// TIA Portal project "Project10" (V15.1)

(* hardware
DEVICE "S71500/ET200MP station_1"  S7-1500 station
   slot 0: "Rail_0"  Rack  6ES7 590-1***0-0AA0
   slot 1: "PLC_1"  CPU 1511C-1 PN  6ES7 511-1CK00-0AB0  V2.6
      slot 3: "CPU display_1"  6ES7591-1AA00-0AA0
DEVICE "HMI_1"  TP700 Comfort
   slot 0: "HMI_1"  TP700 Comfort  6AV2 124-0GC01-0AX0  15.1.0.0
   slot 1: "HMI_RT_1"  TP700 Comfort  6AV2 124-0GC01-0AX0  15.1.0.0
   slot 5: "HMI_1.IE_CP_1"  PROFINET Interface  15.0.1.0
      slot 1: "PROFINET Interface_1"  PROFINET Interface
         slot 1: "Port_1"  Port
         slot 2: "Port_2"  Port
   slot 7: "HMI_1.MPI/DP_CP_1"  MPI/DP Interface  15.0.1.0
*)

// ===== PLC "PLC_1"  CPU 1511C-1 PN =====

VAR_GLOBAL   // PLC tag table "Default tag table"
   "Allow_instrybutor" AT %M500.5 : Bool;
   "Tag_1" AT %I0.1 : Bool;
   "tag_test" AT %I0.2 : Bool;
   "Tag_2" AT %M1.1 : Bool;
END_VAR

DATA_BLOCK "CompareLoginPassword_DB"   // DB1
{ S7_Optimized_Access := 'TRUE' }
VERSION : 0.1
// stored: InstanceOfName CompareLoginPassword
"CompareLoginPassword"
BEGIN
END_DATA_BLOCK

DATA_BLOCK "HMI"   // DB2
{ S7_Optimized_Access := 'TRUE' }
VERSION : 0.1
   VAR
      User_Struct_1 : Struct
         login : Int := 1111;
         password : Int := 1111;
         fuel_amount : Int := 50;
      END_STRUCT;
      User_Struct_2 : Struct
         login : Int := 555;
         password : Int := 555;
         fuel_amount : Int;
      END_STRUCT;
      User_Struct_3 : Struct
         login : Int := 352;
         password : Int := 523;
         fuel_amount : Int;
      END_STRUCT;
      User_Struct_4 : Struct
         login : Int := 568;
         password : Int := 8568;
         fuel_amount : Int;
      END_STRUCT;
      User_Struct_5 : Struct
         login : Int := 5665;
         password : Int := 6555;
         fuel_amount : Int;
      END_STRUCT;
      User_Struct_6 : Struct
         login : Int := 5343;
         password : Int := 1234;
         fuel_amount : Int;
      END_STRUCT;
      User_Struct_7 : Struct
         login : Int := 3321;
         password : Int := 5453;
         fuel_amount : Int;
      END_STRUCT;
      User_Struct_8 : Struct
         login : Int := 6233;
         password : Int := 6433;
         fuel_amount : Int;
      END_STRUCT;
      User_Struct_9 : Struct
         login : Int := 612;
         password : Int := 1253;
         fuel_amount : Int;
      END_STRUCT;
      User_Struct_10 : Struct
         login : Int := 1213;
         password : Int := 1235;
         fuel_amount : Int;
      END_STRUCT;
      HMI_Login_Int : Int;
      HMI_Password_Int : Int;
      HMI_Button_Pressed : Bool;
      HMI_Access_Granted : Bool;
      HMI_Fuel_Amount : Int;
      HMI_Screen_Access : Int;
      filled_value : Int;
      WWW_Tag : Int;
      memory : Int := 1500;
   END_VAR
BEGIN
END_DATA_BLOCK

DATA_BLOCK "instrybutor_DB"   // DB4
{ S7_Optimized_Access := 'TRUE' }
VERSION : 0.1
// stored: InstanceOfName instrybutor
"instrybutor"
BEGIN
END_DATA_BLOCK

// folder: System blocks/Program resources

DATA_BLOCK "IEC_Timer_0_DB"   // DB3
{ S7_Optimized_Access := 'TRUE' }
AUTHOR : Simatic
FAMILY : IEC
NAME : IEC_TMR
VERSION : 1.0
// stored: InstanceOfName IEC_TIMER
"IEC_TIMER"
BEGIN
END_DATA_BLOCK

// folder: (top level)

FUNCTION_BLOCK "CompareLoginPassword"   // FB1, LAD
{ S7_Optimized_Access := 'TRUE' }
VERSION : 0.1
BEGIN

REGION Network 1
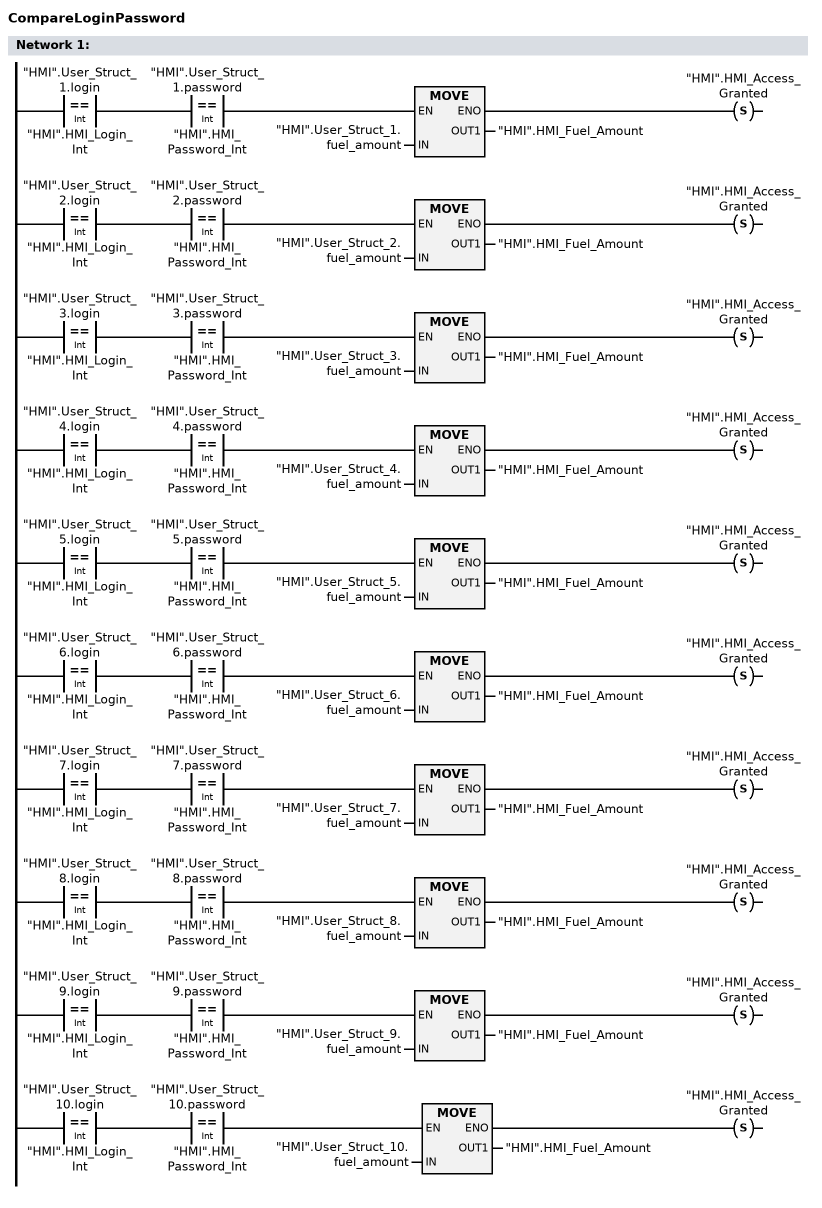
   RUNG wire#powerrail
      { S7_Templates := "SrcType := Int" } EQ_Contact(in1 := "HMI".User_Struct_1.login, in2 := "HMI".HMI_Login_Int)
      { S7_Templates := "SrcType := Int" } EQ_Contact(in1 := "HMI".User_Struct_1.password, in2 := "HMI".HMI_Password_Int)
      Move(in := "HMI".User_Struct_1.fuel_amount, out1 => "HMI".HMI_Fuel_Amount)
      S_Coil( "HMI".HMI_Access_Granted )
   END_RUNG
   RUNG wire#powerrail
      { S7_Templates := "SrcType := Int" } EQ_Contact(in1 := "HMI".User_Struct_2.login, in2 := "HMI".HMI_Login_Int)
      { S7_Templates := "SrcType := Int" } EQ_Contact(in1 := "HMI".User_Struct_2.password, in2 := "HMI".HMI_Password_Int)
      Move(in := "HMI".User_Struct_2.fuel_amount, out1 => "HMI".HMI_Fuel_Amount)
      S_Coil( "HMI".HMI_Access_Granted )
   END_RUNG
   RUNG wire#powerrail
      { S7_Templates := "SrcType := Int" } EQ_Contact(in1 := "HMI".User_Struct_3.login, in2 := "HMI".HMI_Login_Int)
      { S7_Templates := "SrcType := Int" } EQ_Contact(in1 := "HMI".User_Struct_3.password, in2 := "HMI".HMI_Password_Int)
      Move(in := "HMI".User_Struct_3.fuel_amount, out1 => "HMI".HMI_Fuel_Amount)
      S_Coil( "HMI".HMI_Access_Granted )
   END_RUNG
   RUNG wire#powerrail
      { S7_Templates := "SrcType := Int" } EQ_Contact(in1 := "HMI".User_Struct_4.login, in2 := "HMI".HMI_Login_Int)
      { S7_Templates := "SrcType := Int" } EQ_Contact(in1 := "HMI".User_Struct_4.password, in2 := "HMI".HMI_Password_Int)
      Move(in := "HMI".User_Struct_4.fuel_amount, out1 => "HMI".HMI_Fuel_Amount)
      S_Coil( "HMI".HMI_Access_Granted )
   END_RUNG
   RUNG wire#powerrail
      { S7_Templates := "SrcType := Int" } EQ_Contact(in1 := "HMI".User_Struct_5.login, in2 := "HMI".HMI_Login_Int)
      { S7_Templates := "SrcType := Int" } EQ_Contact(in1 := "HMI".User_Struct_5.password, in2 := "HMI".HMI_Password_Int)
      Move(in := "HMI".User_Struct_5.fuel_amount, out1 => "HMI".HMI_Fuel_Amount)
      S_Coil( "HMI".HMI_Access_Granted )
   END_RUNG
   RUNG wire#powerrail
      { S7_Templates := "SrcType := Int" } EQ_Contact(in1 := "HMI".User_Struct_6.login, in2 := "HMI".HMI_Login_Int)
      { S7_Templates := "SrcType := Int" } EQ_Contact(in1 := "HMI".User_Struct_6.password, in2 := "HMI".HMI_Password_Int)
      Move(in := "HMI".User_Struct_6.fuel_amount, out1 => "HMI".HMI_Fuel_Amount)
      S_Coil( "HMI".HMI_Access_Granted )
   END_RUNG
   RUNG wire#powerrail
      { S7_Templates := "SrcType := Int" } EQ_Contact(in1 := "HMI".User_Struct_7.login, in2 := "HMI".HMI_Login_Int)
      { S7_Templates := "SrcType := Int" } EQ_Contact(in1 := "HMI".User_Struct_7.password, in2 := "HMI".HMI_Password_Int)
      Move(in := "HMI".User_Struct_7.fuel_amount, out1 => "HMI".HMI_Fuel_Amount)
      S_Coil( "HMI".HMI_Access_Granted )
   END_RUNG
   RUNG wire#powerrail
      { S7_Templates := "SrcType := Int" } EQ_Contact(in1 := "HMI".User_Struct_8.login, in2 := "HMI".HMI_Login_Int)
      { S7_Templates := "SrcType := Int" } EQ_Contact(in1 := "HMI".User_Struct_8.password, in2 := "HMI".HMI_Password_Int)
      Move(in := "HMI".User_Struct_8.fuel_amount, out1 => "HMI".HMI_Fuel_Amount)
      S_Coil( "HMI".HMI_Access_Granted )
   END_RUNG
   RUNG wire#powerrail
      { S7_Templates := "SrcType := Int" } EQ_Contact(in1 := "HMI".User_Struct_9.login, in2 := "HMI".HMI_Login_Int)
      { S7_Templates := "SrcType := Int" } EQ_Contact(in1 := "HMI".User_Struct_9.password, in2 := "HMI".HMI_Password_Int)
      Move(in := "HMI".User_Struct_9.fuel_amount, out1 => "HMI".HMI_Fuel_Amount)
      S_Coil( "HMI".HMI_Access_Granted )
   END_RUNG
   RUNG wire#powerrail
      { S7_Templates := "SrcType := Int" } EQ_Contact(in1 := "HMI".User_Struct_10.login, in2 := "HMI".HMI_Login_Int)
      { S7_Templates := "SrcType := Int" } EQ_Contact(in1 := "HMI".User_Struct_10.password, in2 := "HMI".HMI_Password_Int)
      Move(in := "HMI".User_Struct_10.fuel_amount, out1 => "HMI".HMI_Fuel_Amount)
      S_Coil( "HMI".HMI_Access_Granted )
   END_RUNG
   // the same network as SCL:
   IF ("HMI".User_Struct_1.login = "HMI".HMI_Login_Int) AND ("HMI".User_Struct_1.password = "HMI".HMI_Password_Int) THEN
       "HMI".HMI_Fuel_Amount := "HMI".User_Struct_1.fuel_amount;
       "HMI".HMI_Access_Granted := TRUE;
   END_IF;
   IF ("HMI".User_Struct_2.login = "HMI".HMI_Login_Int) AND ("HMI".User_Struct_2.password = "HMI".HMI_Password_Int) THEN
       "HMI".HMI_Fuel_Amount := "HMI".User_Struct_2.fuel_amount;
       "HMI".HMI_Access_Granted := TRUE;
   END_IF;
   IF ("HMI".User_Struct_3.login = "HMI".HMI_Login_Int) AND ("HMI".User_Struct_3.password = "HMI".HMI_Password_Int) THEN
       "HMI".HMI_Fuel_Amount := "HMI".User_Struct_3.fuel_amount;
       "HMI".HMI_Access_Granted := TRUE;
   END_IF;
   IF ("HMI".User_Struct_4.login = "HMI".HMI_Login_Int) AND ("HMI".User_Struct_4.password = "HMI".HMI_Password_Int) THEN
       "HMI".HMI_Fuel_Amount := "HMI".User_Struct_4.fuel_amount;
       "HMI".HMI_Access_Granted := TRUE;
   END_IF;
   IF ("HMI".User_Struct_5.login = "HMI".HMI_Login_Int) AND ("HMI".User_Struct_5.password = "HMI".HMI_Password_Int) THEN
       "HMI".HMI_Fuel_Amount := "HMI".User_Struct_5.fuel_amount;
       "HMI".HMI_Access_Granted := TRUE;
   END_IF;
   IF ("HMI".User_Struct_6.login = "HMI".HMI_Login_Int) AND ("HMI".User_Struct_6.password = "HMI".HMI_Password_Int) THEN
       "HMI".HMI_Fuel_Amount := "HMI".User_Struct_6.fuel_amount;
       "HMI".HMI_Access_Granted := TRUE;
   END_IF;
   IF ("HMI".User_Struct_7.login = "HMI".HMI_Login_Int) AND ("HMI".User_Struct_7.password = "HMI".HMI_Password_Int) THEN
       "HMI".HMI_Fuel_Amount := "HMI".User_Struct_7.fuel_amount;
       "HMI".HMI_Access_Granted := TRUE;
   END_IF;
   IF ("HMI".User_Struct_8.login = "HMI".HMI_Login_Int) AND ("HMI".User_Struct_8.password = "HMI".HMI_Password_Int) THEN
       "HMI".HMI_Fuel_Amount := "HMI".User_Struct_8.fuel_amount;
       "HMI".HMI_Access_Granted := TRUE;
   END_IF;
   IF ("HMI".User_Struct_9.login = "HMI".HMI_Login_Int) AND ("HMI".User_Struct_9.password = "HMI".HMI_Password_Int) THEN
       "HMI".HMI_Fuel_Amount := "HMI".User_Struct_9.fuel_amount;
       "HMI".HMI_Access_Granted := TRUE;
   END_IF;
   IF ("HMI".User_Struct_10.login = "HMI".HMI_Login_Int) AND ("HMI".User_Struct_10.password = "HMI".HMI_Password_Int) THEN
       "HMI".HMI_Fuel_Amount := "HMI".User_Struct_10.fuel_amount;
       "HMI".HMI_Access_Granted := TRUE;
   END_IF;
END_REGION
END_FUNCTION_BLOCK

FUNCTION_BLOCK "instrybutor"   // FB2, LAD
{ S7_Optimized_Access := 'TRUE' }
VERSION : 0.1
BEGIN

REGION Network 1
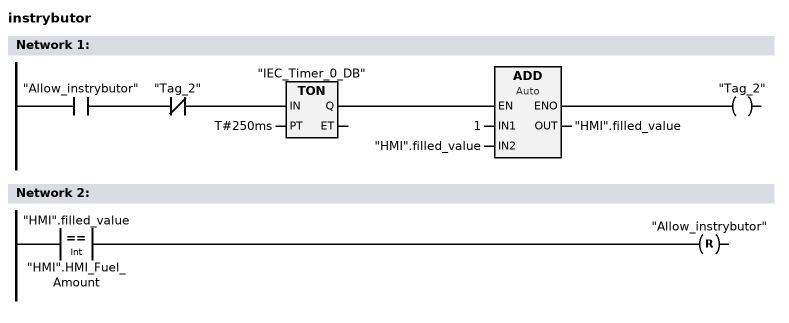
   "IEC_Timer_0_DB".TON(IN := "Allow_instrybutor" AND NOT "Tag_2", PT := T#250ms);
   IF "IEC_Timer_0_DB".Q THEN "HMI".filled_value := 1 + "HMI".filled_value; END_IF;
   "Tag_2" := "IEC_Timer_0_DB".Q;
END_REGION

REGION Network 2
   RUNG wire#powerrail
      { S7_Templates := "SrcType := Int" } EQ_Contact(in1 := "HMI".filled_value, in2 := "HMI".HMI_Fuel_Amount)
      R_Coil( "Allow_instrybutor" )
   END_RUNG
   // the same network as SCL:
   IF "HMI".filled_value = "HMI".HMI_Fuel_Amount THEN "Allow_instrybutor" := FALSE; END_IF;
END_REGION
END_FUNCTION_BLOCK

ORGANIZATION_BLOCK "Main"   // OB1, LAD, ProgramCycle
TITLE = "Main Program Sweep (Cycle)"
{ S7_Optimized_Access := 'TRUE' }
VERSION : 0.1
   VAR_INPUT
      Initial_Call : Bool;   // Initial call of this OB
      Remanence : Bool;   // =True, if remanent data are available
   END_VAR
BEGIN

REGION Network 1
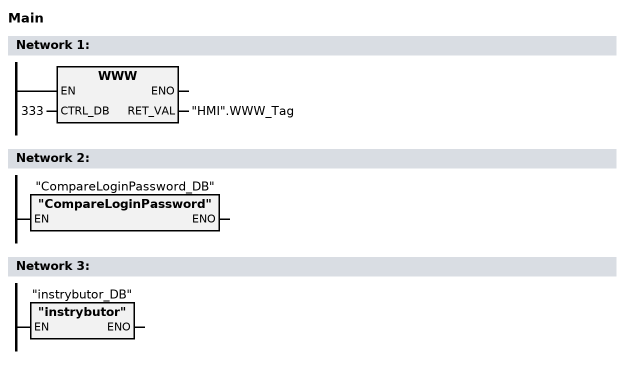
   "HMI".WWW_Tag := WWW(CTRL_DB := 333);
END_REGION

REGION Network 2
   RUNG wire#powerrail
      "CompareLoginPassword_DB"()
   END_RUNG
   // the same network as SCL:
   "CompareLoginPassword_DB"();   // "CompareLoginPassword"
END_REGION

REGION Network 3
   RUNG wire#powerrail
      "instrybutor_DB"()
   END_RUNG
   // the same network as SCL:
   "instrybutor_DB"();   // "instrybutor"
END_REGION
END_ORGANIZATION_BLOCK

(* ===== HMI "HMI_RT_1" =====
system functions are stored by id; their names below are inferred from use
connection "HMI_Connection_1": ETHERNET, S7_1500_OMS

HMI tags "Default tag table"
   "Tag_ScreenNumber" : UInt, internal
   "HMI_Login_Input" : Int = PLC HMI.HMI_Login_Int, 1 s
   "HMI_Password_Input" : Int = PLC HMI.HMI_Password_Int, 1 s
   "HMI_HMI_Access_Granted" : Bool = PLC HMI.HMI_Access_Granted, 1 s
   "Allow_instrybutor" : Bool = PLC Allow_instrybutor AT %M500.5, 1 s
   "HMI_filled_value" : Int = PLC HMI.filled_value, 1 s
   "HMI_HMI_Fuel_Amount" : Int = PLC HMI.HMI_Fuel_Amount, 1 s
   "HMI_WWW_Tag" : Int = PLC HMI.WWW_Tag, 1 s
   "HMI_HMI_Button_Pressed" : Bool = PLC HMI.HMI_Button_Pressed, 1 s

screen "Root screen" 800x420, template "Template_1"
   on GenerateScreen: SetTag("Tag_ScreenNumber", 1)
   TextField "Text field_1" at 147,97 size 117x23; Text 'LOGIN CODE'
   TextField "Text field_2" at 276,97 size 163x23; Text 'PASSWORD CODE'
   IOField "I/O field_1" at 149,130 size 96x32; FormatPattern 99999
      ProcessValue <- "HMI_Login_Input"
   IOField "I/O field_2" at 276,129 size 96x33; FormatPattern 99999
      ProcessValue <- "HMI_Password_Input"
   Button "Button_1" at 215,205 size 96x32; TextOff 'LOGIN'
      on Click: InvertBit("HMI_HMI_Button_Pressed"); SetTag("Tag_ScreenNumber", 2); ActivateScreen("fuel_pump_screen", 0)
      Visibility <- "HMI_HMI_Access_Granted"

Template "Template_1" 800x420
   Button "Exit" at 720,360 size 78x58; TextOff 'Exit'; PictureOff "ExitRuntime_TP700_Comfort_TR"; PictureOn "ExitRuntime_TP700_Comfort_TR"
      on Release: StopRuntime(0)
   Button "Template_Button" at 640,360 size 78x58; TextOff 'Text'
   Button "Template_Button_1" at 560,360 size 78x58; TextOff 'Text'
   Button "Template_Button_2" at 480,360 size 78x58; TextOff 'Text'
   Button "Template_Button_3" at 400,360 size 78x58; TextOff 'Text'
   Button "Template_Button_4" at 321,360 size 78x58; TextOff 'Text'
   Button "Template_Button_5" at 241,360 size 78x58; TextOff 'Text'
   Button "Template_Button_6" at 161,360 size 78x58; TextOff 'Text'
   Button "Alarms" at 81,360 size 78x58; TextOff 'Alarms'; PictureOff "AlarmDisplay_TP700_Comfort_TR"; PictureOn "AlarmDisplay_TP700_Comfort_TR"
      on Release: function_ef3f5d25("Alarm window_Unacknowledged", -1)
   Button "Start screen" at 1,360 size 78x58; TextOff 'Start screen'; PictureOff "NavigateHome_TP700_Comfort_TR"; PictureOn "NavigateHome_TP700_Comfort_TR"
      on Release: ActivateScreen("Root screen", 0)

screen "fuel_pump_screen" 800x420
   on GenerateScreen: SetTag("Tag_ScreenNumber", 2)
   TextField "Text field_1" at 68,39 size 206x33; Text 'ILOŚĆ PALIWA'
   IOField "I/O field_1" at 103,88 size 96x32; FormatPattern 999
      ProcessValue <- "HMI_HMI_Fuel_Amount"
   Button "Button_1" at 685,370 size 96x32; TextOff 'Logout'
      on Click: ResetBit("HMI_HMI_Button_Pressed"); SetTag("HMI_Login_Input", 0); SetTag("HMI_Password_Input", 0); ResetBit("HMI_HMI_Access_Granted"); function_efd93a16(); SetTag("HMI_filled_value", 0)
   Bar "Bar_1" at 591,68 size 80x230; MinimumValue 0; MaximumValue 100
      ProcessValue <- "HMI_filled_value"
      MaximumValue <- "HMI_HMI_Fuel_Amount"
   Button "Button_2" at 50,149 size 218x32; TextOff 'Rozpocznij tankowanie'
      on Click: SetBit("Allow_instrybutor")
*)